{attribute 'qualified_only'}
{attribute 'strict'}
TYPE E_PIDOptimizationStage :
(
	Init,
	RampingUp,
	RampingDown,
	Done
);
END_TYPE

(* stored: Version 1.1.0.1, ProductVersion 3.1.4022.16
   DUT E_PIDOptimizationStage: Id {1ed0394c-f211-4304-974d-674b78c6be4b} *)
